// TIA Portal V19 export
TYPE "PositioningMachine_COut"
// stored: Access Published
   STRUCT
      Infeed_ReqON : Bool;
      CtrlSafe : Bool;
      AxisInOperation : Bool;
      Standstill : Bool;
      InPosition : Bool;
      Bwd_CheckNext : Bool;
      Fwd_CheckNext : Bool;
      VelFwd_VelZero : Bool;
      VelFwd_Running : Bool;
      VelBwd_VelZero : Bool;
      VelBwd_Running : Bool;
      PosBwd_Running : Bool;
      PosFwd_Running : Bool;
      BwdMinusLsSwReached : Bool;   // Bwd / Minus software limit switch reached
      FwdPlusLsSwReached : Bool;   // Fwd / Plus software limit switch reached
      BwdMinusLimitReached : Bool;   // Bwd / Minus external limit reached
      FwdPlusLimitReached : Bool;   // Fwd / Plus software limit reached
      ActualPosition : LReal;
      ActualTargetPos : LReal;
      MinPosition : LReal;   // Actual Fwd / Plus position limit (Software / External)
      MaxPosition : LReal;   // Actual Bwd / Minus position limit (Software / External)
      ActualVelocity : LReal;
      MaxVelocity : LReal;
   END_STRUCT;
END_TYPE
